FUNCTION_BLOCK FB_Sim
VAR_IN_OUT
	Floors:		ARRAY[1..4]	OF	ST_Floor;
	RequestedFloor: INT;
	ActualFloor: INT;

END_VAR
VAR_INPUT
		state:INT;
END_VAR
VAR

	delay3s	:	TON;
	delay6s	:	TON;
END_VAR

CASE State OF
	1:
		Floors[ActualFloor].Mid:=FALSE;
		state:=State+1;
	2:
		Delay3s.IN:=TRUE;
		IF Delay3s.Q THEN
			state:=state+1;
			Delay3s.IN:=FALSE;
		END_IF
	3:
		GVL.Elevator_Y:=GVL.Elevator_Y-55;
		Floors[ActualFloor].High:=TRUE;
		state:=state+1;
	4:
		Delay3s.IN:=TRUE;
		IF Delay3s.Q THEN
			state:=state+1;
			Delay3s.IN:=FALSE;
		END_IF
	5:
		Floors[ActualFloor].High:=FALSE;
		State:=state+1;
	6:
		Delay6s.IN:=TRUE;
		IF Delay6s.Q THEN
			state:=state+1;
			Delay6s.IN:=FALSE;
			ActualFloor:=ActualFloor+1;
		END_IF
	7:
		GVL.Elevator_Y:=GVL.Elevator_Y-71;
		Floors[ActualFloor].Low:=TRUE;
		state:=state+1;
	8:
		Delay3s.IN:=TRUE;
		IF Delay3s.Q THEN
			state:=state+1;
			Delay3s.IN:=FALSE;
		END_IF
	9:
		Floors[ActualFloor].Low:=FALSE;
		state:=state+1;
	
	10:
		Floors[ActualFloor].Mid:=TRUE;
		state:=state+1;
		GVL.Elevator_Y:=GVL.Elevator_Y-55;
	11:	Delay3s.IN:=TRUE;
		IF Delay3s.Q THEN
			state:=1;
			Delay3s.IN:=FALSE;
		END_IF
	12:
		Floors[ActualFloor].Low:=TRUE;
		state:=state+1;
		GVL.Elevator_Y:=GVL.Elevator_Y-71;
	13:
		Delay3s.IN:=TRUE;
		IF Delay3s.Q THEN
			state:=state+1;
			Delay3s.IN:=FALSE;
		END_IF
	14:
		Floors[ActualFloor].Low:=FALSE;
		state:=state+1;
	15:
		GVL.Elevator_Y:=GVL.Elevator_Y-55;
		Floors[ActualFloor].Low:=FALSE;
		Floors[ActualFloor].High:=FALSE;
		Floors[ActualFloor].Mid:=TRUE;
		state:=99;
		
	16:
		Floors[ActualFloor].Mid:=FALSE;
		State:=State+1;
	17:
		Delay3s.IN:=TRUE;
		IF Delay3s.Q THEN
			state:=state+1;
			Delay3s.IN:=FALSE;
		END_IF
	18:
		Floors[ActualFloor].Low:=TRUE;
		GVL.Elevator_Y:=GVL.Elevator_Y+55;
		state:=state+1;
	
	19:
		Delay3s.IN:=TRUE;
		IF Delay3s.Q THEN
			state:=state+1;
			Delay3s.IN:=FALSE;
		END_IF
	
	20:
		Floors[ActualFloor].Low:=FALSE;
		state:=state+1;
	21:
		Delay6s.IN:=TRUE;
		IF Delay6s.Q THEN
			state:=state+1;
			ActualFloor:=ActualFloor-1;
			
			Delay6s.IN:=FALSE;
		END_IF
	22:
		GVL.Elevator_Y:=GVL.Elevator_Y+71;
		Floors[ActualFloor].High:=TRUE;
		state:=state+1;
	
	23:
		Delay3s.IN:=TRUE;
		IF Delay3s.Q THEN
			state:=state+1;
			Delay3s.IN:=FALSE;
		END_IF
	24:
		Floors[ActualFloor].High:=FALSE;
		GVL.Elevator_Y:=GVL.Elevator_Y+55;
		state:=state+1;
	25:
	Floors[ActualFloor].Mid:=TRUE;
	state:=state+1;	
	
	26:
		Delay3s.IN:=TRUE;
		IF Delay3s.Q THEN
			state:=16;
			Delay3s.IN:=FALSE;
		END_IF
		
	27:
		Floors[ActualFloor].High:=TRUE;
		GVL.Elevator_Y:=GVL.Elevator_Y+71;
		state:=state+1;
	28:
		Delay3s.IN:=TRUE;
		IF Delay3s.Q THEN
			state:=state+1;
			Delay3s.IN:=FALSE;
		END_IF
	29:
		Floors[ActualFloor].High:=FALSE;
		state:=state+1;
	30:
		GVL.Elevator_Y:=GVL.Elevator_Y+55;
		Floors[ActualFloor].Low:=FALSE;
		Floors[ActualFloor].High:=FALSE;
		Floors[ActualFloor].Mid:=TRUE;
		state:=99;	
	
END_CASE

delay3s(IN:= delay3s.IN, PT:= T#500MS, Q=> , ET=> );
delay6s(IN:= delay6s.IN, PT:= T#2S, Q=> , ET=> );

END_FUNCTION_BLOCK

(* stored: Version 1.1.0.1, ProductVersion 3.1.4024.9
   POU FB_Sim: Id {85c3bc2d-d7cc-4588-b189-b607db4c79eb}, SpecialFunc None *)
